// TwinCAT 3 PLC project PlcTcProberTests
// Title: PlcTcProberTests
// Company: Vortex.Library
// ProjectVersion: 0.6.0.913
// ProgramVersion: 3.1.4023.0
// libraries:
//   Tc2_Standard, * (Beckhoff Automation GmbH)
//   Tc2_System, * (Beckhoff Automation GmbH)
//   Tc3_Module, * (Beckhoff Automation GmbH)
// project tree:
//   GVLs/ Tests.TcGVL
//   / PlcTask.TcTTO
//   POUs/ MAIN.TcPOU
//   Runners/ fbBasicRunnerTests.TcPOU, fbRecorderRunnerTests.TcPOU, stRecorder.TcDUT
//   Runners/TestStructs/nestedInheritance/ fbInheritanceLevel_1.TcPOU, fbInheritanceLevel_2.TcPOU, fbInheritanceLevel_3.TcPOU, fbInheritanceLevel_4.TcPOU, fbInheritanceLevel_5.TcPOU, fbRootLevelStruct.TcPOU
//   Runners/TestStructs/ stAllTypes.TcDUT
// real-time tasks:
//   TASK PlcTask: cycle T#10ms, priority 20, ADS port 350

CONFIGURATION PlcTcProberTests
    RESOURCE PLC ON TwinCAT3
        TASK PlcTask(INTERVAL := T#10ms, PRIORITY := 20);
        PROGRAM MAIN WITH PlcTask : MAIN;
    END_RESOURCE
END_CONFIGURATION

// ---- Runners/stRecorder.TcDUT
TYPE stRecorder :
STRUCT
    counter : INT;
END_STRUCT
END_TYPE

// ---- Runners/TestStructs/stAllTypes.TcDUT
{attribute addProperty Interpolated "|[[2]AttributeName]|-|[[1]AttributeName]|-|[AttributeName]||[BOOL_val.AttributeName]|"}
{attribute addProperty Name "ALL BASE TYPES"}
TYPE stAllTypes :
STRUCT
    {attribute addProperty Name "BOOL"}
    BOOL_val : BOOL;
    {attribute addProperty Name "BYTE"}
    BYTE_val : BYTE; //   0-255 8 bit
    {attribute addProperty Name "WORD"}
    WORD_val : WORD; //   0-65535 16 bit
    {attribute addProperty Name "DWORD"}
    DWORD_val : DWORD; //   0-4294967295 32 bit
    {attribute addProperty Name "LWORD"}
    LWORD_val : LWORD; //   0-264-1 64 bit
    {attribute addProperty Name "SINT"}
    SINT_val : SINT; //   -128-127 8 bit
    {attribute addProperty Name "USINT"}
    USINT_val : USINT; //   0-255 8 bit
    {attribute addProperty Name "INT"}
    INT_val : INT; //   -32768-32767 16 bit
    {attribute addProperty Name "UINT"}
    UINT_val : UINT; //   0-65535 16 bit
    {attribute addProperty Name "DINT"}
    DINT_val : DINT; //   -2147483648-2147483647 32 bit
    {attribute addProperty Name "UDINT"}
    UDINT_val : UDINT; //   0-4294967295 32 bit
    {attribute addProperty Name "LINT"}
    LINT_val : LINT; //   -263-263-1 64 bit
    {attribute addProperty Name "ULINT"}
    ULINT_val : ULINT; //   0-264-1 64 bit
    {attribute addProperty Name "REAL"}
    REAL_val : REAL; //   -3.402823E+38-3.402823E+38 32 bit
    {attribute addProperty Name "LREAL"}
    LREAL_val : LREAL; //   -1.7976931348623158e+308-1.7976931348623158e+308 64 bit
    {attribute addProperty Name "STRING(82)"}
    STRING_val : STRING; //   -
    {attribute addProperty Name "WSTRING(82)"}
    WSTRING_val : WSTRING; //   -
    {attribute addProperty Name "TIME"}
    TIME_val : TIME; //   0-4294967295 32 bit
    {attribute addProperty Name "TIME OF DAY"}
    TIME_OF_DAY_val : TIME_OF_DAY; //   0 (00:00:00:000)-4294967295 (23:59:59:999) 32 bit
    {attribute addProperty Name "DATE"}
    DATE_val : DATE; //   0 (01.01.1970)-4294967295 (7 February 2106) 32 bit
    {attribute addProperty Name "DATE TIME"}
    DATE_AND_TIME_val : DATE_AND_TIME; //   0 (01.01.1970, 00:00)-4294967295 (7 February 2106, 6:28:15) 32 bit
    {attribute addProperty Name "TOD"}
    TOD_val : TOD; //   0 (00:00:00:000)-4294967295 (23:59:59:999) 32 bit
    {attribute addProperty Name "DT"}
    DT_val : DT; //   0 (01.01.1970, 00:00)-4294967295 (7 February 2106, 6:28:15) 32 bit
    {attribute addProperty Name "LTIME"}
    LTIME_val : LTIME; //   0-213503d23h34m33s709ms551us615ns 64 bit
    {attribute addProperty Name "ARRAY OF BASE TYPES"}
    ValueTypeArray : ARRAY[0..5, 0..3, 0..2] OF INT;
END_STRUCT
END_TYPE

// ---- GVLs/Tests.TcGVL
{attribute 'qualified_only'}
VAR_GLOBAL
    _basicRunnerTests : fbBasicRunnerTests;
    _recorderRunnerTests : fbRecorderRunnerTests;
END_VAR

// ---- POUs/MAIN.TcPOU
PROGRAM MAIN
VAR
    InheritanceRw : fbInheritanceLevel_5;
END_VAR

END_PROGRAM

// ---- Runners/TestStructs/nestedInheritance/fbInheritanceLevel_5.TcPOU
FUNCTION_BLOCK fbInheritanceLevel_5 EXTENDS fbInheritanceLevel_4
VAR
    {attribute addProperty Name "LEVEL 5"}
    level_5 : stAllTypes;
END_VAR

METHOD Init : BOOL
VAR_INPUT
END_VAR
SUPER^.Init();
END_METHOD

END_FUNCTION_BLOCK

// ---- Runners/TestStructs/nestedInheritance/fbInheritanceLevel_4.TcPOU
FUNCTION_BLOCK fbInheritanceLevel_4 EXTENDS fbInheritanceLevel_3
VAR
    {attribute addProperty Name "LEVEL 4"}
    level_4 : stAllTypes;
END_VAR

SUPER^();

METHOD Init : BOOL
VAR_INPUT
END_VAR
SUPER^.Init();
END_METHOD

END_FUNCTION_BLOCK

// ---- Runners/TestStructs/nestedInheritance/fbInheritanceLevel_3.TcPOU
FUNCTION_BLOCK fbInheritanceLevel_3 EXTENDS fbInheritanceLevel_2
VAR
    {attribute addProperty Name "LEVEL 3"}
    level_3 : stAllTypes;
END_VAR

SUPER^();

METHOD Init : BOOL
VAR_INPUT
END_VAR
SUPER^.Init();
END_METHOD

END_FUNCTION_BLOCK

// ---- Runners/TestStructs/nestedInheritance/fbInheritanceLevel_2.TcPOU
FUNCTION_BLOCK fbInheritanceLevel_2 EXTENDS fbInheritanceLevel_1
VAR
    {attribute addProperty Name "LEVEL 2"}
    level_2 : stAllTypes;
END_VAR

SUPER^();

METHOD Init : BOOL
VAR_INPUT
END_VAR
SUPER^.Init();
END_METHOD

END_FUNCTION_BLOCK

// ---- Runners/TestStructs/nestedInheritance/fbInheritanceLevel_1.TcPOU
FUNCTION_BLOCK fbInheritanceLevel_1 EXTENDS fbRootLevelStruct
VAR
    {attribute addProperty Name "LEVEL 1"}
    level_1 : stAllTypes;
END_VAR

SUPER^();

{attribute 'obsolete' := 'Use method Initialize() instead'}
METHOD Init : BOOL
VAR_INPUT
END_VAR
SUPER^.Init();
level_1.BYTE_val := 255;
level_1.WORD_val := 65535;
level_1.DWORD_val := 4294967295;
level_1.LWORD_val := 18446744073709551615;
level_1.SINT_val := 127;
level_1.USINT_val := 255;
level_1.INT_val := 32767;
level_1.UINT_val := 65535;
level_1.DINT_val := 2147483647;
level_1.UDINT_val := 4294967295;
level_1.LINT_val := 9223372036854775807;
level_1.ULINT_val := 18446744073709551615;
level_1.REAL_val := 3.402823E+38;
level_1.LREAL_val := 1.7976931348623158E+308;
level_1.STRING_val := 'ABCDEFGHIJKLMNOPRSTUWZ';
level_1.WSTRING_val := "fdalsdflahsdjhfajksdry9837489";
level_1.TIME_val := T#1H;
level_1.TIME_OF_DAY_val := TOD#23:59:59.999;
level_1.DATE_val := DATE#2106-02-07;
level_1.DATE_AND_TIME_val := DT#2106-02-07-6:28:15;
level_1.TOD_val := TOD#23:59:59.999;
level_1.DT_val := DT#2106-02-07-6:28:15;
level_1.LTIME_val := LTIME#213503D23H34M33S709MS551US615NS;
END_METHOD

END_FUNCTION_BLOCK

// ---- Runners/TestStructs/nestedInheritance/fbRootLevelStruct.TcPOU
FUNCTION_BLOCK fbRootLevelStruct
VAR
    {attribute addProperty Name "LEVEL 0"}
    level_0 : stAllTypes;
END_VAR
VAR CONSTANT
    level : INT := 5;
END_VAR

METHOD Init : BOOL
VAR_INPUT
END_VAR
level_0.BYTE_val := 0;
level_0.WORD_val := 0;
level_0.DWORD_val := 0;
level_0.LWORD_val := 0;
level_0.SINT_val := -128;
level_0.USINT_val := 0;
level_0.INT_val := -32768;
level_0.UINT_val := 0;
level_0.DINT_val := -2147483648;
level_0.UDINT_val := 0;
level_0.LINT_val := -9223372036854775808;
level_0.ULINT_val := 0;
level_0.REAL_val := -3.402823E+38;
level_0.LREAL_val := -1.7976931348623158E+308;
level_0.STRING_val := '';
level_0.WSTRING_val := "";
level_0.TIME_val := T#0S;
level_0.TIME_OF_DAY_val := TOD#00:00:00.000;
level_0.DATE_val := DATE#1970-01-01;
level_0.DATE_AND_TIME_val := DT#1970-01-01-00:00;
level_0.TOD_val := TOD#00:00:00.000;
level_0.DT_val := DT#1970-01-01-00:00;
level_0.LTIME_val := LTIME#0S;
END_METHOD

END_FUNCTION_BLOCK

// ---- Runners/fbBasicRunnerTests.TcPOU
FUNCTION_BLOCK fbBasicRunnerTests
VAR
    runs : UINT;
END_VAR

{attribute 'TcRpcEnable'}
METHOD ResetCounter : UINT
runs := 0;
END_METHOD

{attribute 'TcRpcEnable'}
METHOD RunCount : UINT
runs := runs + 1;
RunCount := runs;
END_METHOD

{attribute 'TcRpcEnable'}
METHOD RunUntilReturnsTrue : BOOL
VAR_INPUT
    _m : BOOL;
END_VAR
RunUntilReturnsTrue := _m;
END_METHOD

END_FUNCTION_BLOCK

// ---- Runners/fbRecorderRunnerTests.TcPOU
FUNCTION_BLOCK fbRecorderRunnerTests
VAR
    _recorder : stRecorder;
END_VAR

{attribute 'TcRpcEnable'}
METHOD ResetCounter : UINT
_recorder.counter := 0;
END_METHOD

{attribute 'TcRpcEnable'}
METHOD RunWithRecorder : INT
RunWithRecorder := _recorder.counter;
END_METHOD

END_FUNCTION_BLOCK
